FUNCTION_BLOCK ACTUORSbutton
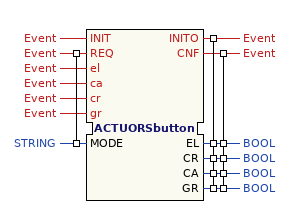
  EVENT_INPUT
    INIT;
    REQ WITH MODE;
    el;
    ca;
    cr;
    gr;
  END_EVENT
  EVENT_OUTPUT
    INITO WITH EL, CA, CR, GR;
    CNF WITH EL, CA, CR, GR;
  END_EVENT
  VAR_INPUT
    MODE : STRING;
  END_VAR
  VAR_OUTPUT
    EL : BOOL;
    CR : BOOL;
    CA : BOOL;
    GR : BOOL;
  END_VAR
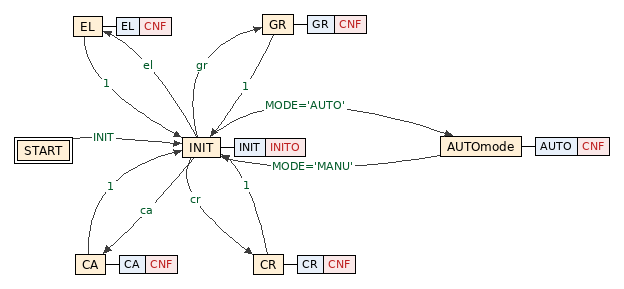
  EC_STATES
    START;
    INIT : INIT -> INITO;
    EL : EL -> CNF;
    CA : CA -> CNF;
    CR : CR -> CNF;
    GR : GR -> CNF;
    AUTOmode : AUTO -> CNF;
  END_STATES
  EC_TRANSITIONS
    START TO INIT := INIT;
    EL TO INIT := 1;
    GR TO INIT := 1;
    CA TO INIT := 1;
    CR TO INIT := 1;
    INIT TO EL := el;
    INIT TO GR := gr;
    INIT TO CA := ca;
    INIT TO CR := cr;
    INIT TO AUTOmode := MODE='AUTO';
    AUTOmode TO INIT := MODE='MANU';
  END_TRANSITIONS
  ALGORITHM INIT IN ST:
CA := FALSE;
EL := FALSE;
CR := FALSE;
GR := FALSE;
  END_ALGORITHM
  ALGORITHM EL IN ST:
EL := TRUE;
  END_ALGORITHM
  ALGORITHM CA IN ST:
CA := TRUE;
  END_ALGORITHM
  ALGORITHM CR IN ST:
CR := TRUE;
  END_ALGORITHM
  ALGORITHM GR IN ST:
GR := TRUE;
  END_ALGORITHM
  ALGORITHM AUTO IN ST:
CA := TRUE;
EL := TRUE;
CR := TRUE;
GR := TRUE;
  END_ALGORITHM
END_FUNCTION_BLOCK
